PROGRAM MAIN
VAR
	// Create by Huang Hansheng 2019.09.14
	fbGenerator			: FB_Generator;
	fbGeneratorEx		:FB_GeneratorEx;
	iGenerator			:IGenerator;
	bChange				:BOOL;
	_tCycleTime			:TIME:= T#2S;
	sVendor				:STRING;
	bOutput				:BOOL;
END_VAR

IF	bChange THEN 
	iGenerator := fbGenerator;
ELSE
	iGenerator := fbGeneratorEx;
END_IF

iGenerator.P_tCycleTime :=  _tCycleTime;

bOutput :=  iGenerator.Flash();

sVendor := iGenerator.P_Vendor;

END_PROGRAM

(* stored: Version 1.1.0.1, ProductVersion 3.1.4022.16
   POU MAIN: Id {33a74080-58f5-4de8-85c4-f45ae5c1cfc0}, SpecialFunc None *)
